// TIA Portal project "S7-1500 için Lojik Ve-Veya-Özel Veya-Tersleme Komutu" (V18)

(* hardware
DEVICE "S7-1500/ET200MP station_1"  S7-1500 station
   slot 0: "Rail_0"  Rack  6ES7 590-1***0-0AA0
   slot 1: "PLC_1"  CPU 1512C-1 PN  6ES7 512-1CK00-0AB0  V2.8
      slot 3: "CPU display_1"  6ES7591-1AA00-0AA0
      slot 32768: "PROFINET interface_1"  X1
         slot 32769: "Port_1"  X1 P1
         slot 32770: "Port_2"  X1 P2
      slot 34817: "Virtual CP interface port_1"  Virtual CP interface port  Virtual CP interface port
*)

// ===== PLC "PLC_1"  CPU 1512C-1 PN =====

VAR_GLOBAL   // PLC tag table "Default tag table"
   "Tag_1" AT %I0.0 : Bool;
   "Tag_2" AT %MW10 : Int;
   "Tag_3" AT %Q0.0 : Bool;
   "Tag_4" AT %I0.1 : Bool;
   "Tag_5" AT %Q0.1 : Bool;
   "Tag_6" AT %MW11 : Int;
   "Tag_7" AT %MW12 : Int;
   "Tag_8" AT %MW13 : Int;
   "Tag_9" AT %MW14 : Int;
   "Tag_10" AT %I0.2 : Bool;
   "Tag_11" AT %I0.3 : Bool;
END_VAR

ORGANIZATION_BLOCK "Main"   // OB1, LAD, ProgramCycle
TITLE = "Main Program Sweep (Cycle)"
{ S7_Optimized_Access := 'TRUE' }
VERSION : 0.1
   VAR_INPUT
      Initial_Call : Bool;   // Initial call of this OB
      Remanence : Bool;   // =True, if remanent data are available
   END_VAR
BEGIN

REGION Network 1: 5 ve 10 un binary değerleri verilmiş. Aynı satırda olanlara "Ve(AND)" uygular ve sonucu MW10'a yazar.
   // 5 =0101
   // 10=1010 
   // -------------------
   // Sonuç==>0000 yani sonuç 0 olur.
   // Simülasyonda 16 tabanında sonuç veriyor. Bunu çözmek için simülasyon çalışırken AND kapısına sağ tık yapıp Modify-->Display Format-->Decimal yapmak lazım.
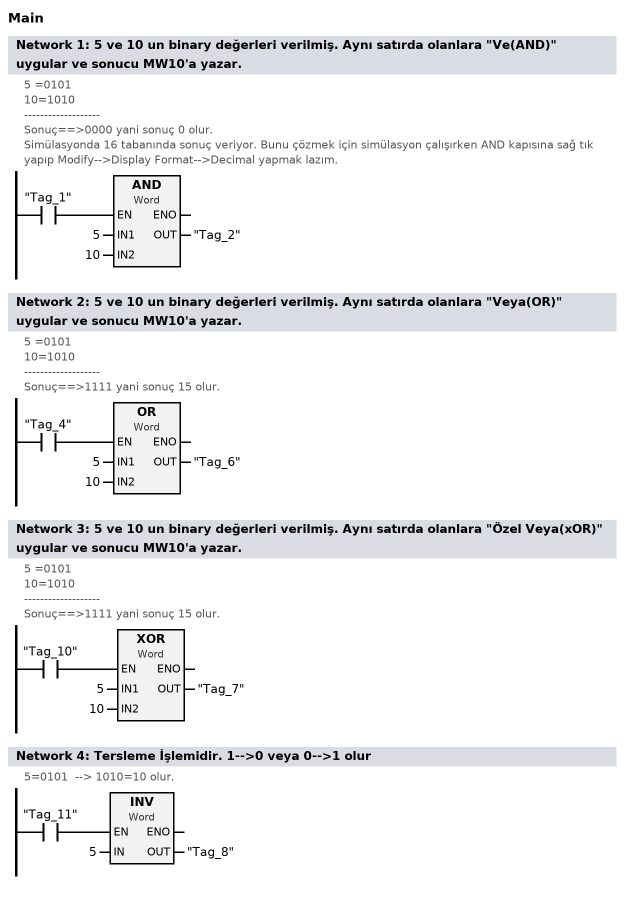
   RUNG wire#powerrail
      Contact( "Tag_1" )
      { S7_Templates := "SrcType := Word" } And(in1 := 5, in2 := 10, out => "Tag_2")
   END_RUNG
   // the same network as SCL:
   IF "Tag_1" THEN "Tag_2" := 5 AND 10; END_IF;
END_REGION

REGION Network 2: 5 ve 10 un binary değerleri verilmiş. Aynı satırda olanlara "Veya(OR)" uygular ve sonucu MW10'a yazar.
   // 5 =0101
   // 10=1010 
   // -------------------
   // Sonuç==>1111 yani sonuç 15 olur.
   IF "Tag_4" THEN "Tag_6" := 5 OR 10; END_IF;
END_REGION

REGION Network 3: 5 ve 10 un binary değerleri verilmiş. Aynı satırda olanlara "Özel Veya(xOR)" uygular ve sonucu MW10'a yazar.
   // 5 =0101
   // 10=1010 
   // -------------------
   // Sonuç==>1111 yani sonuç 15 olur.
   IF "Tag_10" THEN "Tag_7" := 5 XOR 10; END_IF;
END_REGION

REGION Network 4: Tersleme İşlemidir. 1-->0 veya 0-->1 olur
   // 5=0101  --> 1010=10 olur.
   RUNG wire#powerrail
      Contact( "Tag_11" )
      { S7_Templates := "SrcType := Word" } Inv(in := 5, out => "Tag_8")
   END_RUNG
   // the same network as SCL:
   IF "Tag_11" THEN "Tag_8" := NOT 5; END_IF;
END_REGION
END_ORGANIZATION_BLOCK